// TwinCAT 3 PLC project Runtime
// ProgramVersion: 3.1.4023.0
// libraries:
//   Tc2_Standard, * (Beckhoff Automation GmbH)
//   Tc2_System, * (Beckhoff Automation GmbH)
//   Tc3_Module, * (Beckhoff Automation GmbH)
// project tree:
//   / E_States.TcDUT, FB_Motor.TcPOU, MAIN.TcPOU, PlcTask.TcTTO, ST_LevelSensors.TcDUT
// real-time tasks:
//   TASK PlcTask: cycle T#20ms, priority 20, ADS port 350
// I/O:
//   DEVICE Device 1 (EtherCAT) (disabled), AmsNetId 169.254.141.45.2.1
//     Term 1 (EK1100) [EK1100 EtherCAT Coupler (2A E-Bus)]
//       Term 2 (EL1809) [EL1809 16Ch. Dig. Input 24V, 3ms]
//       Term 3 (EL2004) [EL2004 4Ch. Dig. Output 24V, 0.5A]
// variable links:
//   Runtime/Runtime Instance <-> Device 1 (EtherCAT)/Term 1 (EK1100)/Term 2 (EL1809)
//     PlcTask Inputs/MAIN.BT_FloorCall[1] <-> Channel 10/Input
//     PlcTask Inputs/MAIN.BT_FloorCall[2] <-> Channel 11/Input
//     PlcTask Inputs/MAIN.BT_FloorCall[3] <-> Channel 12/Input
//     PlcTask Inputs/MAIN.LS_Floor[1].High <-> Channel 3/Input
//     PlcTask Inputs/MAIN.LS_Floor[2].High <-> Channel 6/Input
//     PlcTask Inputs/MAIN.LS_Floor[3].High <-> Channel 9/Input
//     PlcTask Inputs/MAIN.LS_Floor[1].Low <-> Channel 1/Input
//     PlcTask Inputs/MAIN.LS_Floor[2].Low <-> Channel 4/Input
//     PlcTask Inputs/MAIN.LS_Floor[3].Low <-> Channel 7/Input
//     PlcTask Inputs/MAIN.LS_Floor[1].Mid <-> Channel 2/Input
//     PlcTask Inputs/MAIN.LS_Floor[2].Mid <-> Channel 5/Input
//     PlcTask Inputs/MAIN.LS_Floor[3].Mid <-> Channel 8/Input
//   Runtime/Runtime Instance <-> Device 1 (EtherCAT)/Term 1 (EK1100)/Term 3 (EL2004)
//     PlcTask Outputs/MAIN.Elevator.Brake <-> Channel 4/Output
//     PlcTask Outputs/MAIN.Elevator.Down <-> Channel 2/Output
//     PlcTask Outputs/MAIN.Elevator.Slow <-> Channel 3/Output
//     PlcTask Outputs/MAIN.Elevator.Up <-> Channel 1/Output

CONFIGURATION Runtime
    RESOURCE PLC ON TwinCAT3
        TASK PlcTask(INTERVAL := T#20ms, PRIORITY := 20);
        PROGRAM MAIN WITH PlcTask : MAIN;
    END_RESOURCE
END_CONFIGURATION

// ---- E_States.TcDUT
{attribute 'qualified_only'}
{attribute 'strict'}
TYPE E_States :
(
	Call := 0,//same as idle state
	MoveUp,
	MoveDown,
	IncrementFloor,
	DecrementFloor,
	SlowDown,
	Stop
);
END_TYPE

// ---- ST_LevelSensors.TcDUT
TYPE ST_LevelSensors :
STRUCT
	Low,
	Mid,
	High AT %I*:BOOL;
END_STRUCT
END_TYPE

// ---- MAIN.TcPOU
PROGRAM MAIN
VAR
	LS_Floor:ARRAY[1..3]	OF	ST_LevelSensors;
	BT_FloorCall AT %I*:ARRAY[1..3]	OF	BOOL;
	Elevator:FB_Motor;
	STATE: E_States;
	RequestedFloor: INT;
	i: INT;
	CurrentFloor: INT;
	PulseTrigger:ARRAY[1..3]OF	TP;
	LatchTime: ULINT;
	ElapsedTime: LTIME;
END_VAR


CASE STATE	OF	
	E_States.Call:;
		//action logic
		FOR	i:=1 TO 3	DO
			IF	BT_FloorCall[i]	THEN
				RequestedFloor:=i;
				LatchTime:=F_GetSystemTime();
				EXIT;
			END_IF
		END_FOR
		//transitions
		IF	RequestedFloor>CurrentFloor	THEN
			STATE:=E_States.MoveUp;
		ELSIF	RequestedFloor<CurrentFloor	THEN
			STATE:=E_States.MoveDown;
		END_IF
		
		//initialise pulse timer
		FOR	i:=1	TO	3	DO
			PulseTrigger[i](IN:=FALSE);
		END_FOR
		
	E_States.MoveUp:
		Elevator.MoveUp();
		FOR	i:=1	TO	3	DO
			PulseTrigger[i](IN:=LS_Floor[i].Low,PT:=T#10MS);
			IF	PulseTrigger[i].Q	THEN
				STATE:=E_States.IncrementFloor;
			END_IF
		END_FOR
		IF	RequestedFloor=CurrentFloor	THEN	
			state:=E_States.SlowDown;
		END_IF
		
	E_States.MoveDown:
		Elevator.MoveDown();
		FOR	i:=1	TO	3	DO
			PulseTrigger[i](IN:=LS_Floor[i].High,PT:=T#10MS);
			IF	PulseTrigger[i].Q	THEN
				STATE:=E_States.DecrementFloor;
			END_IF
		END_FOR
		IF	RequestedFloor=CurrentFloor	THEN	
			state:=E_States.SlowDown;
		END_IF
		
	E_States.IncrementFloor:
		CurrentFloor:=CurrentFloor+1;
		STATE:=E_States.MoveUp;
	E_States.DecrementFloor:
		CurrentFloor:=CurrentFloor-1;
		STATE:=E_States.MoveDown;
	E_States.SlowDown:
		Elevator.SlowDown();
		FOR	i:=1	TO	3	DO
			IF	LS_Floor[i].Mid	THEN
				STATE:=E_States.Stop;
			END_IF
		END_FOR
	E_States.Stop:
		//ElapsedTime:=ULINT_TO_LTIME(F_GetSystemTime()-LatchTime);
		Elevator.Stop();
		state:=E_States.Call;
END_CASE

END_PROGRAM

// ---- FB_Motor.TcPOU
FUNCTION_BLOCK FB_Motor
VAR_INPUT
END_VAR
VAR_OUTPUT
END_VAR
VAR
	Up,
	Down,
	Slow ,
	Brake AT %Q* :BOOL;
END_VAR

ACTION MoveDown:
Up:=FALSE;
Down:=TRUE;
Slow:=FALSE;

Brake:=FALSE;
END_ACTION

ACTION MoveUp:
Up:=TRUE;
Down:=FALSE;
Slow:=FALSE;

Brake:=FALSE;
END_ACTION

ACTION SlowDown:
Slow:=TRUE;
END_ACTION

ACTION Stop:
Up:=FALSE;
Down:=FALSE;
Slow:=FALSE;
Brake:=TRUE;
END_ACTION

END_FUNCTION_BLOCK
